//上下出=2
IF Autoflow=1
	AND AutoStatus
	AND NOT(DisablePB[11])
	AND LS_S11_UpDownBack
	AND NOT(SOL_S11_UpDown)
	AND (MachineRunStatus AND NOT(IndexData[11].FinishFlag[11]) AND IndexData[11].FinishFlag[10] AND IndexData[11].OKFlag[10] AND NOT(IndexData[11].NGFlag[10])
	OR Rtrig_test.Q) THEN
	Autoflow:=2;
	Error_LS_S11_UpDownOut1:=FALSE;
END_IF;
TON1(In:=Autoflow=2 AND LS_S11_UpDownOut, PT:=t#500ms);
//檢查開始=3
IF Autoflow=2 AND TON1.Q THEN
	Autoflow:=3;
END_IF;
IF Autoflow=3 AND HMIPV_S11_CurrentValue<=HMISV_S11_MaxValue AND HMIPV_S11_CurrentValue>=HMISV_S11_MinValue THEN		//OK
	IndexData[11].OKFlag[11]:=TRUE;
	IndexData[11].NGFlag[11]:=FALSE;
	IndexData[11].ErrorLog[11]:=0;
END_IF;
IF Autoflow=3 AND (HMIPV_S11_CurrentValue>HMISV_S11_MaxValue OR HMIPV_S11_CurrentValue<HMISV_S11_MinValue) THEN		//NG
	Error_LS_S11_UpDownOut1:=TRUE;
	IndexData[11].OKFlag[11]:=FALSE;
	IndexData[11].NGFlag[11]:=TRUE;
	IndexData[11].ErrorLog[11]:=3;
	BatchIndexCount:=BatchIndexCount-1;
END_IF;
TON2(In:=Autoflow=3 AND IndexData[11].FinishFlag[11], PT:=t#1000ms);
//上下回=4
IF Autoflow=3 AND TON2.Q AND (Rtrig_test.Q OR NOT(StepMode)) THEN
	Autoflow:=4;
END_IF;

//*************************************************************************
//手動
//上下電磁閥
R_TRIG_1[0](CLK:=HMIPB_SOL_S11_UpDown AND NOT(AutoStatus));
interlockback[0]:=TRUE;
interlockout[0]:=SNR_Index AND NOT(RY_Index);
(*SET*)
IF ((R_TRIG_1[0].Q AND NOT(solstatus[0])) OR Autoflow=2) AND interlockout[0] THEN
	SOL_S11_UpDown:=TRUE;
END_IF;
(*RESET*)
IF ((R_TRIG_1[0].Q AND (solstatus[0])) OR Autoflow=4 OR Initflow=4) AND interlockback[0] THEN
	SOL_S11_UpDown:=FALSE;
END_IF;
(*STATUS*)
solstatus[0]:=SOL_S11_UpDown;

//標準值設定
IF HMIPB_S11_StandarValueSet THEN
	HMISV_S11_StandarValue:=HMIPV_S11_CurrentValue;
END_IF;

HMISV_S11_MaxValue:=HMISV_S11_StandarValue+HMISV_S11_PValue;	//最大值
HMISV_S11_MinValue:=HMISV_S11_StandarValue-HMISV_S11_NValue;	//最小值

(*************************************************************************
程序名稱:第11站檢查上夾板RESET流程
作者:蔡相偉
版本,日期,版本資訊:
1.0.0		2017/11/22		初始版本

PowerOn=0
Idle=1
上下回=4
*************************************************************************)
//PowerOn=0
IF NOT(SystemReadyStatus) THEN
	Initflow:=0;
END_IF;

//Idle=1
IF Initflow=0 AND SystemReadyStatus THEN
	Initflow:=1;
END_IF;

IF Initflow=4 AND LS_S11_UpDownBack THEN
	Initflow:=1;
END_IF;

//上下回=4
F_TRIG_1(CLK:= ErrorStatus[11] OR Error_PB_Estop);
IF Initflow=1 AND (F_TRIG_1.Q OR Manual2AutoFlag) THEN
	Initflow:=4;
END_IF;

//*************************************************************************
//Cycle Time
//*************************************************************************
TON_CT(In:=AutoFlow>1, PT:=t#500s);
CycleTime[11]:=LINT_TO_DINT(TimeToSec( TON_CT.ET));
END_PROGRAM

PROGRAM prStation13
VAR
    interlockback : ARRAY[0..1] OF BOOL;
    interlockout : ARRAY[0..1] OF BOOL;
    solstatus : ARRAY[0..1] OF BOOL;
    R_TRIG_1 : ARRAY[0..1] OF R_TRIG;
    Rtrig_test : R_TRIG;
    F_TRIG_1 : F_TRIG;
    Autoflow : INT;
    Initflow : INT;
    TON1 : TON;
    TON2 : TON;
    tPressTime : TIME;
    TON_CT : TON;
END_VAR
VAR_EXTERNAL
    IndexData : ARRAY[0..19] OF stIndexData;
    DisablePB : ARRAY[0..19] OF BOOL;
    SystemReadyStatus : BOOL;
    AutoStatus : BOOL;
    ErrorStatus : ARRAY[0..19] OF BOOL;
    Error_PB_EStop : BOOL;
    LS_S13_UpDownBack : BOOL;
    MachineRunStatus : BOOL;
    LS_S13_UpDownOut : BOOL;
    HMIPB_SOL_S13_UpDown : BOOL;
    SNR_Index : BOOL;
    RY_Index : BOOL;
    SOL_S13_UpDown : BOOL;
    Manual2AutoFlag : BOOL;
    TestPB : ARRAY[0..19] OF BOOL;
    LS_S13_TempHighWarring : BOOL;
    LS_S13_TempLowWarring : BOOL;
    Error_LS_S13_TempHighWarring : BOOL;
    Error_LS_S13_TempLowWarring : BOOL;
    HMISV_S13_PressTime : DINT;
    CycleTime : ARRAY[0..19] OF DINT;
    BatchIndexCount : DINT;
    Error_LS_S11_UpDownOut1 : BOOL;
    Error_LS_S13_UpDownOut1 : BOOL;
    StepMode : BOOL;
END_VAR
(*************************************************************************
程序名稱:第13站壓合流程
作者:蔡相偉
版本,日期,版本資訊:
1.0.0		2017/11/22		初始版本

PowerOn=0
Idle=1
上下出=2
檢查開始=3
上下回=4
*************************************************************************)
(*************************************************************************
異常碼
急停=1
氣缸=2
檢查NG=3
*************************************************************************)
//*************************************************************************
//本站狀態判斷
IF IndexData[13].OKFlag[13]
	OR IndexData[13].NGFlag[13] THEN
	IndexData[13].FinishFlag[13]:=TRUE;
END_IF;
//前站狀態判斷
IF  	IndexData[13].NGFlag[11] THEN
	IndexData[13].NGFlag[11]:=TRUE;
END_IF;
//本站關閉判斷
IF DisablePB[13] AND IndexData[13].FinishFlag[11] AND IndexData[13].OKFlag[11] AND NOT(IndexData[13].NGFlag[11]) THEN
	IndexData[13].OKFlag[13]:=TRUE;
END_IF;

Rtrig_test(CLK:=TestPB[13]);
//PowerOn=0
IF NOT(SystemReadyStatus AND AutoStatus AND NOT(ErrorStatus[13]) AND NOT(Error_PB_EStop)) THEN
	Autoflow:=0;
END_IF;
	//EStop異常碼
	IF Error_PB_Estop AND NOT(IndexData[13].FinishFlag[13]) AND IndexData[13].OkFlag[1] THEN
		IndexData[13].NGFlag[13]:=TRUE;
		IndexData[13].ErrorLog[13]:=1;
		BatchIndexCount:=BatchIndexCount-1;
	END_IF;
	//Error異常碼
	IF ErrorStatus[13] AND NOT(IndexData[13].FinishFlag[13]) AND IndexData[13].OkFlag[1] THEN
		IndexData[13].NGFlag[13]:=TRUE;
		IndexData[13].ErrorLog[13]:=2;
		BatchIndexCount:=BatchIndexCount-1;
	END_IF;
//Idle=1
IF AutoFlow=0 AND SystemReadyStatus AND AutoStatus AND NOT(ErrorStatus[13]) AND NOT(Error_PB_EStop) THEN
	AutoFlow:=1;
END_IF;

IF Autoflow=4 AND LS_S13_UpDownBack THEN
	Autoflow:=1;
END_IF;

//上下出=2
IF Autoflow=1
	AND AutoStatus
	AND NOT(DisablePB[13])
	AND LS_S13_UpDownBack
	AND NOT(SOL_S13_UpDown)
	AND NOT(Error_LS_S13_TempHighWarring)
	AND NOT(Error_LS_S13_TempLowWarring)
	AND (MachineRunStatus AND NOT(IndexData[13].FinishFlag[13]) AND IndexData[13].FinishFlag[11] AND IndexData[13].OKFlag[11] AND NOT(IndexData[13].NGFlag[11])
	OR Rtrig_test.Q) THEN
	Autoflow:=2;
	Error_LS_S13_UpDownOut1:=FALSE;
END_IF;

//檢查開始=3
IF Autoflow=2 AND NOT(LS_S13_UpDownBack) THEN
	Autoflow:=3;
END_IF;
tPressTime:=NanoSecToTime(HMISV_S13_PressTime*100000000);	//Define
TON1(In:=Autoflow=3 AND LS_S13_UpDownOut, PT:=tPressTime);		//OK
TON2(In:=NOT(TON1.Q), PT:=t#2s);		//NG
//上下回=4
IF Autoflow=3 AND TON1.Q AND (Rtrig_test.Q OR NOT(StepMode)) THEN
	IndexData[13].OKFlag[13]:=TRUE;
	IndexData[13].NGFlag[13]:=FALSE;
	IndexData[13].ErrorLog[13]:=0;
	Autoflow:=4;
END_IF;

IF Autoflow=3 AND TON2.Q AND (Rtrig_test.Q OR NOT(StepMode)) THEN
	Error_LS_S13_UpDownOut1:=TRUE;
	IndexData[13].OKFlag[13]:=FALSE;
	IndexData[13].NGFlag[13]:=TRUE;
	IndexData[13].ErrorLog[13]:=3;
	BatchIndexCount:=BatchIndexCount-1;
	Autoflow:=4;
END_IF;

//*************************************************************************
//手動
//上下電磁閥
R_TRIG_1[0](CLK:=HMIPB_SOL_S13_UpDown AND NOT(AutoStatus));
interlockback[0]:=TRUE;
interlockout[0]:=SNR_Index AND NOT(RY_Index);
(*SET*)
IF ((R_TRIG_1[0].Q AND NOT(solstatus[0])) OR Autoflow=2) AND interlockout[0] THEN
	SOL_S13_UpDown:=TRUE;
END_IF;
(*RESET*)
IF ((R_TRIG_1[0].Q AND (solstatus[0])) OR Autoflow=4 OR Initflow=4) AND interlockback[0] THEN
	SOL_S13_UpDown:=FALSE;
END_IF;
(*STATUS*)
solstatus[0]:=SOL_S13_UpDown;
(*************************************************************************
程序名稱:第13站壓合RESET流程
作者:蔡相偉
版本,日期,版本資訊:
1.0.0		2017/11/22		初始版本

PowerOn=0
Idle=1
上下回=4
*************************************************************************)
//PowerOn=0
IF NOT(SystemReadyStatus) THEN
	Initflow:=0;
END_IF;

//Idle=1
IF Initflow=0 AND SystemReadyStatus THEN
	Initflow:=1;
END_IF;

IF Initflow=4 AND LS_S13_UpDownBack THEN
	Initflow:=1;
END_IF;

//上下回=4
F_TRIG_1(CLK:= ErrorStatus[13] OR Error_PB_Estop);
IF Initflow=1 AND (F_TRIG_1.Q OR Manual2AutoFlag) THEN
	Initflow:=4;
END_IF;

//*************************************************************************
//Cycle Time
//*************************************************************************
TON_CT(In:=AutoFlow>1, PT:=t#500s);
CycleTime[13]:=LINT_TO_DINT(TimeToSec( TON_CT.ET));
END_PROGRAM

PROGRAM prStation15
VAR
    interlockback : ARRAY[0..1] OF BOOL;
    interlockout : ARRAY[0..1] OF BOOL;
    solstatus : ARRAY[0..1] OF BOOL;
    R_TRIG_1 : ARRAY[0..1] OF R_TRIG;
    Rtrig_test : R_TRIG;
    F_TRIG_1 : F_TRIG;
    Autoflow : INT;
    Initflow : INT;
    TON1 : TON;
    TON2 : TON;
    TON_CT : TON;
END_VAR
VAR_EXTERNAL
    IndexData : ARRAY[0..19] OF stIndexData;
    DisablePB : ARRAY[0..19] OF BOOL;
    SystemReadyStatus : BOOL;
    AutoStatus : BOOL;
    ErrorStatus : ARRAY[0..19] OF BOOL;
    Error_PB_EStop : BOOL;
    MachineRunStatus : BOOL;
    SNR_Index : BOOL;
    RY_Index : BOOL;
    Manual2AutoFlag : BOOL;
    TestPB : ARRAY[0..19] OF BOOL;
    HMIPB_SOL_S15_UpDown : BOOL;
    SOL_S15_UpDown : BOOL;
    HMISV_S15_StandarValue : DINT;
    HMIPV_S15_CurrentValue : DINT;
    HMISV_S15_MaxValue : DINT;
    HMISV_S15_PValue : DINT;
    HMISV_S15_MinValue : DINT;
    HMISV_S15_NValue : DINT;
    HMIPB_S15_StandarValueSet : BOOL;
    LS_S15_UpDownBack : BOOL;
    LS_S15_UpDownOut : BOOL;
    CycleTime : ARRAY[0..19] OF DINT;
    BatchIndexCount : DINT;
    Error_LS_S13_UpDownOut1 : BOOL;
    Error_LS_S15_UpDownOut1 : BOOL;
    StepMode : BOOL;
END_VAR
(*************************************************************************
程序名稱:第15站檢查壓合流程
作者:蔡相偉
版本,日期,版本資訊:
1.0.0		2017/11/28		初始版本

PowerOn=0
Idle=1
上下出=2
檢查開始=3
上下回=4
*************************************************************************)
(*************************************************************************
異常碼
急停=1
氣缸=2
檢查NG=3
*************************************************************************)
//*************************************************************************
//本站狀態判斷
IF IndexData[15].OKFlag[15]
	OR IndexData[15].NGFlag[15] THEN
	IndexData[15].FinishFlag[15]:=TRUE;
END_IF;
//前站狀態判斷
IF  	IndexData[15].NGFlag[13] THEN
	IndexData[15].NGFlag[13]:=TRUE;
END_IF;
//本站關閉判斷
IF DisablePB[15] AND IndexData[15].FinishFlag[13] AND IndexData[15].OKFlag[13] AND NOT(IndexData[15].NGFlag[13]) THEN
	IndexData[15].OKFlag[15]:=TRUE;
END_IF;

Rtrig_test(CLK:=TestPB[15]);
//PowerOn=0
IF NOT(SystemReadyStatus AND AutoStatus AND NOT(ErrorStatus[15]) AND NOT(Error_PB_EStop)) THEN
	Autoflow:=0;
END_IF;
	//EStop異常碼
	IF Error_PB_Estop AND NOT(IndexData[15].FinishFlag[15]) AND IndexData[15].OkFlag[1] THEN
		IndexData[15].NGFlag[15]:=TRUE;
		IndexData[15].ErrorLog[15]:=1;
		BatchIndexCount:=BatchIndexCount-1;
	END_IF;
	//Error異常碼
	IF ErrorStatus[15] AND NOT(IndexData[15].FinishFlag[15]) AND IndexData[15].OkFlag[1] THEN
		IndexData[15].NGFlag[15]:=TRUE;
		IndexData[15].ErrorLog[15]:=2;
		BatchIndexCount:=BatchIndexCount-1;
	END_IF;
//Idle=1
IF AutoFlow=0 AND SystemReadyStatus AND AutoStatus AND NOT(ErrorStatus[15]) AND NOT(Error_PB_EStop) THEN
	AutoFlow:=1;
END_IF;

IF Autoflow=4 AND LS_S15_UpDownBack THEN
	Autoflow:=1;
END_IF;

//上下出=2
IF Autoflow=1
	AND AutoStatus
	AND NOT(DisablePB[15])
	AND LS_S15_UpDownBack
	AND NOT(SOL_S15_UpDown)
	AND (MachineRunStatus AND NOT(IndexData[15].FinishFlag[15]) AND IndexData[15].FinishFlag[13] AND IndexData[15].OKFlag[13] AND NOT(IndexData[15].NGFlag[13])
	OR Rtrig_test.Q) THEN
	Autoflow:=2;
	Error_LS_S15_UpDownOut1:=FALSE;
END_IF;
TON1(In:=Autoflow=2 AND LS_S15_UpDownOut, PT:=t#500ms);
//檢查開始=3
IF Autoflow=2 AND TON1.Q THEN
	Autoflow:=3;
END_IF;
IF Autoflow=3 AND NOT(IndexData[15].FinishFlag[15]) AND HMIPV_S15_CurrentValue<=HMISV_S15_MaxValue AND HMIPV_S15_CurrentValue>=HMISV_S15_MinValue THEN		//OK
	IndexData[15].OKFlag[15]:=TRUE;
	IndexData[15].NGFlag[15]:=FALSE;
	IndexData[15].ErrorLog[15]:=0;
END_IF;
IF Autoflow=3 AND NOT(IndexData[15].FinishFlag[15]) AND (HMIPV_S15_CurrentValue>HMISV_S15_MaxValue OR HMIPV_S15_CurrentValue<HMISV_S15_MinValue) THEN		//NG
	Error_LS_S15_UpDownOut1:=TRUE;
	IndexData[15].OKFlag[15]:=FALSE;
	IndexData[15].NGFlag[15]:=TRUE;
	IndexData[15].ErrorLog[15]:=3;
	BatchIndexCount:=BatchIndexCount-1;
END_IF;
TON2(In:=Autoflow=3 AND IndexData[15].FinishFlag[15], PT:=t#1000ms);
//上下回=4
IF Autoflow=3 AND TON2.Q AND (Rtrig_test.Q OR NOT(StepMode)) THEN
	Autoflow:=4;
END_IF;

//*************************************************************************
//手動
//上下電磁閥
R_TRIG_1[0](CLK:=HMIPB_SOL_S15_UpDown AND NOT(AutoStatus));
interlockback[0]:=TRUE;
interlockout[0]:=SNR_Index AND NOT(RY_Index);
(*SET*)
IF ((R_TRIG_1[0].Q AND NOT(solstatus[0])) OR Autoflow=2) AND interlockout[0] THEN
	SOL_S15_UpDown:=TRUE;
END_IF;
(*RESET*)
IF ((R_TRIG_1[0].Q AND (solstatus[0])) OR Autoflow=4 OR Initflow=4) AND interlockback[0] THEN
	SOL_S15_UpDown:=FALSE;
END_IF;
(*STATUS*)
solstatus[0]:=SOL_S15_UpDown;

//標準值設定
IF HMIPB_S15_StandarValueSet THEN
	HMISV_S15_StandarValue:=HMIPV_S15_CurrentValue;
END_IF;

HMISV_S15_MaxValue:=HMISV_S15_StandarValue+HMISV_S15_PValue;	//最大值
HMISV_S15_MinValue:=HMISV_S15_StandarValue-HMISV_S15_NValue;	//最小值

(*************************************************************************
程序名稱:第15站檢查壓合RESET流程
作者:蔡相偉
版本,日期,版本資訊:
1.0.0		2017/11/22		初始版本

PowerOn=0
Idle=1
上下回=4
*************************************************************************)
//PowerOn=0
IF NOT(SystemReadyStatus) THEN
	Initflow:=0;
END_IF;

//Idle=1
IF Initflow=0 AND SystemReadyStatus THEN
	Initflow:=1;
END_IF;

IF Initflow=4 AND LS_S15_UpDownBack THEN
	Initflow:=1;
END_IF;

//上下回=4
F_TRIG_1(CLK:= ErrorStatus[15] OR Error_PB_Estop);
IF Initflow=1 AND (F_TRIG_1.Q OR Manual2AutoFlag) THEN
	Initflow:=4;
END_IF;

//*************************************************************************
//Cycle Time
//*************************************************************************
TON_CT(In:=AutoFlow>1, PT:=t#500s);
CycleTime[15]:=LINT_TO_DINT(TimeToSec( TON_CT.ET));
END_PROGRAM

PROGRAM prStation16
VAR
    AutoFlow : INT;
    Rtrig_test : R_TRIG;
    Rtrig_test2 : R_TRIG;
    TON_CT : TON;
END_VAR
VAR_EXTERNAL
    IndexData : ARRAY[0..19] OF stIndexData;
    DisablePB : ARRAY[0..19] OF BOOL;
    TestPB : ARRAY[0..19] OF BOOL;
    SystemReadyStatus : BOOL;
    ErrorStatus : ARRAY[0..19] OF BOOL;
    Error_PB_EStop : BOOL;
    AutoStatus : BOOL;
    MachineRunStatus : BOOL;
    HMIPB_YAMAHA_Unload_OKStart : BOOL;
    YAMAHA_Unload_OKStart : BOOL;
    YAMAHA_Unload_Finish : BOOL;
    HMIPB_YAMAHA_Unload_NGStart : BOOL;
    YAMAHA_Unload_NGStart : BOOL;
    CycleTime : ARRAY[0..19] OF DINT;
    BatchOKCount : DINT;
    BatchIndexCount : DINT;
    BatchNGCount : DINT;
END_VAR
(*
程序名稱:第16站下料流程
作者:蔡相偉
版本,日期,版本資訊:
1.0.0		2017/11/21		初始版本
PowerOn=0
Idle=1|--->OK下料開始=10--->OK下料完成=11
		  |--->NG下料開始=20--->NG下料完成=21
*)
//本站狀態判斷
IF IndexData[16].OKFlag[16]
	OR IndexData[16].NGFlag[16] THEN
	IndexData[16].FinishFlag[16]:=TRUE;
END_IF;

//前站狀態判斷
IF NOT(IndexData[16].OKFlag[1]) THEN
	IndexData[16].NGFlag[16]:=TRUE;
END_IF;

(*
//本站關閉判斷
IF DisablePB[1] THEN
	IndexData[1].NGFlag[1]:=TRUE;
END_IF;
*)
Rtrig_test(CLK:=HMIPB_YAMAHA_Unload_OKStart);
Rtrig_test2(CLK:=HMIPB_YAMAHA_Unload_NGStart);
//PowerOn=0
IF NOT(SystemReadyStatus AND AutoStatus AND NOT(ErrorStatus[16]) AND NOT(Error_PB_EStop)) THEN
	Autoflow:=0;
END_IF;

//Idle=1
IF AutoFlow=0 AND SystemReadyStatus AND AutoStatus AND NOT(ErrorStatus[16]) AND NOT(Error_PB_EStop) THEN
	AutoFlow:=1;
END_IF;

IF AutoFlow=11 AND NOT(YAMAHA_Unload_OKStart) AND IndexData[16].FinishFlag[16] THEN
	AutoFlow:=1;
END_IF;

IF AutoFlow=21 AND NOT(YAMAHA_Unload_NGStart) AND IndexData[16].FinishFlag[16] THEN
	AutoFlow:=1;
END_IF;

//OK下料開始=10
IF Autoflow=1
	AND AutoStatus
	AND NOT(DisablePB[16])
	AND (MachineRunStatus AND NOT(IndexData[16].FinishFlag[16]) AND IndexData[16].OKFlag[1] AND IndexData[16].FinishFlag[15] AND IndexData[16].OKFlag[15] AND NOT(IndexData[16].NGFlag[15]) OR Rtrig_test.Q) THEN
	Autoflow:=10;
END_IF;
IF AutoFlow=10 THEN
	YAMAHA_Unload_OKStart:=TRUE;
END_IF;
IF YAMAHA_Unload_Finish OR AutoFlow=0 THEN
	YAMAHA_Unload_OKStart:=FALSE;
END_IF;

//OK下料完成=11
IF AutoFlow=10 AND (YAMAHA_Unload_Finish) THEN
	BatchOKCount:=BatchOKCount+1;
	BatchIndexCount:=BatchIndexCount-1;
	AutoFlow:=11;
END_IF;
IF AutoFlow=11 THEN
	IndexData[16].OKFlag[16]:=TRUE;
END_IF;

//NG下料開始=20
IF Autoflow=1
	AND AutoStatus
	AND NOT(DisablePB[16])
	AND (MachineRunStatus AND NOT(IndexData[16].FinishFlag[16]) AND IndexData[16].OKFlag[1] AND IndexData[16].FinishFlag[15] AND (IndexData[16].NGFlag[15]) OR Rtrig_test2.Q) THEN
	Autoflow:=20;
END_IF;
IF AutoFlow=20 THEN
	YAMAHA_Unload_NGStart:=TRUE;
END_IF;
IF YAMAHA_Unload_Finish OR AutoFlow=0 THEN
	YAMAHA_Unload_NGStart:=FALSE;
END_IF;

//NG下料完成=21
IF AutoFlow=20 AND (YAMAHA_Unload_Finish) THEN
	BatchNGCount:=BatchNGCount+1;
	BatchIndexCount:=BatchIndexCount-1;
	AutoFlow:=21;
END_IF;
IF AutoFlow=21 THEN
	IndexData[16].NGFlag[16]:=TRUE;
END_IF;

//*************************************************************************
//Cycle Time
//*************************************************************************
TON_CT(In:=AutoFlow>1, PT:=t#500s);
CycleTime[16]:=LINT_TO_DINT(TimeToSec( TON_CT.ET));
END_PROGRAM

PROGRAM prFeedAndSupplier
VAR
    Supplier_S6 : fbFull;
    Supplier_S8 : fbFull;
    Supplier_S10 : fbFull;
    Feeder_S6 : fbFeed;
    Feeder_S8 : fbFeed;
    Feeder_S10 : fbFeed;
END_VAR
VAR_EXTERNAL
    SNR_S6_Full : BOOL;
    RY_S6_Full : BOOL;
    Error_SNR_S6_Full : BOOL;
    FullNotExistTime : ARRAY[0..19] OF DINT;
    FullExistTime : ARRAY[0..19] OF DINT;
    FullNotExistErrorTime : ARRAY[0..19] OF DINT;
    SNR_S8_Full : BOOL;
    RY_S8_Full : BOOL;
    Error_SNR_S8_Full : BOOL;
    SNR_S10_Full : BOOL;
    RY_S10_Full : BOOL;
    Error_SNR_S10_Full : BOOL;
    FeedStart : ARRAY[0..19] OF BOOL;
    PB_Reset : BOOL;
    FeedFinish : ARRAY[0..19] OF BOOL;
    Error_LS_S6_THBack : BOOL;
    Error_LS_S6_THOut : BOOL;
    LS_S6_UpDownBack : BOOL;
    SOL_S6_UpDown : BOOL;
    LS_S6_MoveBack : BOOL;
    SNR_S6_Feed : BOOL;
    LS_S6_THBack : BOOL;
    LS_S6_THOut : BOOL;
    HMIPB_SOL_S6_TH : BOOL;
    FeedNotExistTime : ARRAY[0..19] OF DINT;
    FeedExistTime : ARRAY[0..19] OF DINT;
    Error_SNR_S6_Feed : BOOL;
    RY_S6_Feed : BOOL;
    SOL_S6_TH : BOOL;
    Error_LS_S8_THBack : BOOL;
    Error_LS_S8_THOut : BOOL;
    LS_S8_UpDownBack : BOOL;
    SOL_S8_UpDown : BOOL;
    LS_S8_MoveBack : BOOL;
    SNR_S8_Feed : BOOL;
    LS_S8_THBack : BOOL;
    LS_S8_THOut : BOOL;
    HMIPB_SOL_S8_TH : BOOL;
    Error_SNR_S8_Feed : BOOL;
    RY_S8_Feed : BOOL;
    SOL_S8_TH : BOOL;
    Error_LS_S10_THBack : BOOL;
    Error_LS_S10_THOut : BOOL;
    LS_S10_UpDownBack : BOOL;
    SOL_S10_UpDown : BOOL;
    LS_S10_MoveBack : BOOL;
    SNR_S10_Feed : BOOL;
    LS_S10_THBack : BOOL;
    LS_S10_THOut : BOOL;
    HMIPB_SOL_S10_TH : BOOL;
    Error_SNR_S10_Feed : BOOL;
    RY_S10_Feed : BOOL;
    SOL_S10_TH : BOOL;
    Manual2AutoFlag : BOOL;
END_VAR
//第6站振動筒
Supplier_S6();
Supplier_S6.bFullSNR:=SNR_S6_Full;
Supplier_S6.iItemNotExistDelayTime:=FullNotExistTime[6];
Supplier_S6.iItemExistTime:=FullExistTime[6];
Supplier_S6.iItemNotExistErrorTime:=FullNotExistErrorTime[6];
RY_S6_Full:=Supplier_S6.bFullRY;
Error_SNR_S6_Full:=Supplier_S6.bFullSNRError;

//第8站振動筒
Supplier_S8();
Supplier_S8.bFullSNR:=SNR_S8_Full;
Supplier_S8.iItemNotExistDelayTime:=FullNotExistTime[8];
Supplier_S8.iItemExistTime:=FullExistTime[8];
Supplier_S8.iItemNotExistErrorTime:=FullNotExistErrorTime[8];
RY_S8_Full:=Supplier_S8.bFullRY;
Error_SNR_S8_Full:=Supplier_S8.bFullSNRError;

//第10站振動筒
Supplier_S10();
Supplier_S10.bFullSNR:=SNR_S10_Full;
Supplier_S10.iItemNotExistDelayTime:=FullNotExistTime[10];
Supplier_S10.iItemExistTime:=FullExistTime[10];
Supplier_S10.iItemNotExistErrorTime:=FullNotExistErrorTime[10];
RY_S10_Full:=Supplier_S10.bFullRY;
Error_SNR_S10_Full:=Supplier_S10.bFullSNRError;

//第6站平送
Feeder_S6();
Feeder_S6.bErrorTHBack:=Error_LS_S6_THBack;
Feeder_S6.bErrorTHOut:=Error_LS_S6_THOut;
Feeder_S6.bFeedStart:=FeedStart[6] OR Manual2AutoFlag;
Feeder_S6.bInterlock_thback:=(LS_S6_UpDownBack AND NOT(SOL_S6_UpDown)) OR NOT(LS_S6_MoveBack);
Feeder_S6.bInterlock_thout:=(LS_S6_UpDownBack AND NOT(SOL_S6_UpDown)) OR NOT(LS_S6_MoveBack);
Feeder_S6.bObjSNR:=SNR_S6_Feed;
Feeder_S6.bReset:=PB_Reset;
Feeder_S6.bSupplierRY:=RY_S6_Full;
Feeder_S6.bTHBackLS:=LS_S6_THBack;
Feeder_S6.bTHOutLS:=LS_S6_THOut;
Feeder_S6.bTHPB:=HMIPB_SOL_S6_TH;
Feeder_S6.wNoObjDelayTime:=FeedNotExistTime[6];
Feeder_S6.wObjectExistDelayTime:=FeedExistTime[6];
Error_SNR_S6_Feed :=Feeder_S6.bFeedError;
FeedFinish[6]:= Feeder_S6.bFeedFinish;
RY_S6_Feed:= Feeder_S6.bFeedRY;
SOL_S6_TH:= Feeder_S6.bTHSOL;

//第8站平送
Feeder_S8();
Feeder_S8.bErrorTHBack:=Error_LS_S8_THBack;
Feeder_S8.bErrorTHOut:=Error_LS_S8_THOut;
Feeder_S8.bFeedStart:=FeedStart[8] OR Manual2AutoFlag;
Feeder_S8.bInterlock_thback:=(LS_S8_UpDownBack AND NOT(SOL_S8_UpDown)) OR NOT(LS_S8_MoveBack);
Feeder_S8.bInterlock_thout:=(LS_S8_UpDownBack AND NOT(SOL_S8_UpDown)) OR NOT(LS_S8_MoveBack);
Feeder_S8.bObjSNR:=SNR_S8_Feed;
Feeder_S8.bReset:=PB_Reset;
Feeder_S8.bSupplierRY:=RY_S8_Full;
Feeder_S8.bTHBackLS:=LS_S8_THBack;
Feeder_S8.bTHOutLS:=LS_S8_THOut;
Feeder_S8.bTHPB:=HMIPB_SOL_S8_TH;
Feeder_S8.wNoObjDelayTime:=FeedNotExistTime[8];
Feeder_S8.wObjectExistDelayTime:=FeedExistTime[8];
Error_SNR_S8_Feed:=Feeder_S8.bFeedError;
FeedFinish[8]:= Feeder_S8.bFeedFinish;
RY_S8_Feed:= Feeder_S8.bFeedRY;
SOL_S8_TH:= Feeder_S8.bTHSOL;

//第10站平送
Feeder_S10();
Feeder_S10.bErrorTHBack:=Error_LS_S10_THBack;
Feeder_S10.bErrorTHOut:=Error_LS_S10_THOut;
Feeder_S10.bFeedStart:=FeedStart[10] OR Manual2AutoFlag;
Feeder_S10.bInterlock_thback:=(LS_S10_UpDownBack AND NOT(SOL_S10_UpDown)) OR NOT(LS_S10_MoveBack);
Feeder_S10.bInterlock_thout:=(LS_S10_UpDownBack AND NOT(SOL_S10_UpDown)) OR NOT(LS_S10_MoveBack);
Feeder_S10.bObjSNR:=SNR_S10_Feed;
Feeder_S10.bReset:=PB_Reset;
Feeder_S10.bSupplierRY:=RY_S10_Full;
Feeder_S10.bTHBackLS:=LS_S10_THBack;
Feeder_S10.bTHOutLS:=LS_S10_THOut;
Feeder_S10.bTHPB:=HMIPB_SOL_S10_TH;
Feeder_S10.wNoObjDelayTime:=FeedNotExistTime[10];
Feeder_S10.wObjectExistDelayTime:=FeedExistTime[10];
Error_SNR_S10_Feed:=Feeder_S10.bFeedError;
FeedFinish[10]:= Feeder_S10.bFeedFinish;
RY_S10_Feed:= Feeder_S10.bFeedRY;
SOL_S10_TH:= Feeder_S10.bTHSOL;
END_PROGRAM

PROGRAM prNGCount
VAR
    R_TRIG1 : ARRAY[0..19] OF R_TRIG;
    iCount : ARRAY[0..19] OF INT;
END_VAR
VAR_EXTERNAL
    IndexData : ARRAY[0..19] OF stIndexData;
    Error_NGCount : ARRAY[0..19] OF BOOL;
    PB_Reset : BOOL;
    HMIPB_PB_Reset : BOOL;
END_VAR
//Over 3 times NG S2
R_TRIG1[0](Clk:=IndexData[2].NGFlag[2]);
IF IndexData[2].OKFlag[1] AND R_TRIG1[0].Q THEN
	iCount[2]:=iCount[2]+1;
END_IF;
IF IndexData[2].OKFlag[2] THEN
	iCount[2]:=0;
END_IF;
IF iCount[2]>=3 THEN
	Error_NGCount[2]:=TRUE;
ELSE
	Error_NGCount[2]:=FALSE;
END_IF;
IF PB_Reset OR HMIPB_PB_Reset THEN
	iCount[2]:=0;
END_IF;

//Over 3 times NG S4
R_TRIG1[1](Clk:=IndexData[4].NGFlag[4]);
IF IndexData[4].OKFlag[1] AND R_TRIG1[1].Q THEN
	iCount[4]:=iCount[4]+1;
END_IF;
IF IndexData[4].OKFlag[4] THEN
	iCount[4]:=0;
END_IF;
IF iCount[4]>=3 THEN
	Error_NGCount[4]:=TRUE;
ELSE
	Error_NGCount[4]:=FALSE;
END_IF;
IF PB_Reset OR HMIPB_PB_Reset THEN
	iCount[4]:=0;
END_IF;

//Over 3 times NG S5
R_TRIG1[2](Clk:=IndexData[5].NGFlag[5]);
IF IndexData[5].OKFlag[1] AND R_TRIG1[2].Q THEN
	iCount[5]:=iCount[5]+1;
END_IF;
IF IndexData[5].OKFlag[5] THEN
	iCount[5]:=0;
END_IF;
IF iCount[5]>=3 THEN
	Error_NGCount[5]:=TRUE;
ELSE
	Error_NGCount[5]:=FALSE;
END_IF;
IF PB_Reset OR HMIPB_PB_Reset THEN
	iCount[5]:=0;
END_IF;

//Over 3 times NG S6
R_TRIG1[3](Clk:=IndexData[6].NGFlag[6]);
IF IndexData[6].OKFlag[1] AND R_TRIG1[3].Q THEN
	iCount[6]:=iCount[6]+1;
END_IF;
IF IndexData[6].OKFlag[6] THEN
	iCount[6]:=0;
END_IF;
IF iCount[6]>=3 THEN
	Error_NGCount[6]:=TRUE;
ELSE
	Error_NGCount[6]:=FALSE;
END_IF;
IF PB_Reset OR HMIPB_PB_Reset THEN
	iCount[6]:=0;
END_IF;

//Over 3 times NG S7
R_TRIG1[4](Clk:=IndexData[7].NGFlag[7]);
IF IndexData[7].OKFlag[1] AND R_TRIG1[4].Q THEN
	iCount[7]:=iCount[7]+1;
END_IF;
IF IndexData[7].OKFlag[7] THEN
	iCount[7]:=0;
END_IF;
IF iCount[7]>=3 THEN
	Error_NGCount[7]:=TRUE;
ELSE
	Error_NGCount[7]:=FALSE;
END_IF;
IF PB_Reset OR HMIPB_PB_Reset THEN
	iCount[7]:=0;
END_IF;

//Over 3 times NG S8
R_TRIG1[5](Clk:=IndexData[8].NGFlag[8]);
IF IndexData[8].OKFlag[1] AND R_TRIG1[5].Q THEN
	iCount[8]:=iCount[8]+1;
END_IF;
IF IndexData[8].OKFlag[8] THEN
	iCount[8]:=0;
END_IF;
IF iCount[8]>=3 THEN
	Error_NGCount[8]:=TRUE;
ELSE
	Error_NGCount[8]:=FALSE;
END_IF;
IF PB_Reset OR HMIPB_PB_Reset THEN
	iCount[8]:=0;
END_IF;

//Over 3 times NG S9
R_TRIG1[6](Clk:=IndexData[9].NGFlag[9]);
IF IndexData[9].OKFlag[1] AND R_TRIG1[6].Q THEN
	iCount[9]:=iCount[9]+1;
END_IF;
IF IndexData[9].OKFlag[9] THEN
	iCount[9]:=0;
END_IF;
IF iCount[9]>=3 THEN
	Error_NGCount[9]:=TRUE;
ELSE
	Error_NGCount[9]:=FALSE;
END_IF;
IF PB_Reset OR HMIPB_PB_Reset THEN
	iCount[9]:=0;
END_IF;

//Over 3 times NG S10
R_TRIG1[7](Clk:=IndexData[10].NGFlag[10]);
IF IndexData[10].OKFlag[1] AND R_TRIG1[7].Q THEN
	iCount[10]:=iCount[10]+1;
END_IF;
IF IndexData[10].OKFlag[10] THEN
	iCount[10]:=0;
END_IF;
IF iCount[10]>=3 THEN
	Error_NGCount[10]:=TRUE;
ELSE
	Error_NGCount[10]:=FALSE;
END_IF;
IF PB_Reset OR HMIPB_PB_Reset THEN
	iCount[10]:=0;
END_IF;

//Over 3 times NG S11
R_TRIG1[8](Clk:=IndexData[11].NGFlag[11]);
IF IndexData[11].OKFlag[1] AND R_TRIG1[8].Q THEN
	iCount[11]:=iCount[11]+1;
END_IF;
IF IndexData[11].OKFlag[11] THEN
	iCount[11]:=0;
END_IF;
IF iCount[11]>=3 THEN
	Error_NGCount[11]:=TRUE;
ELSE
	Error_NGCount[11]:=FALSE;
END_IF;
IF PB_Reset OR HMIPB_PB_Reset THEN
	iCount[11]:=0;
END_IF;

//Over 3 times NG S13
R_TRIG1[9](Clk:=IndexData[13].NGFlag[13]);
IF IndexData[13].OKFlag[1] AND R_TRIG1[9].Q THEN
	iCount[13]:=iCount[13]+1;
END_IF;
IF IndexData[13].OKFlag[13] THEN
	iCount[13]:=0;
END_IF;
IF iCount[13]>=3 THEN
	Error_NGCount[13]:=TRUE;
ELSE
	Error_NGCount[13]:=FALSE;
END_IF;
IF PB_Reset OR HMIPB_PB_Reset THEN
	iCount[13]:=0;
END_IF;

//Over 3 times NG S15
R_TRIG1[10](Clk:=IndexData[15].NGFlag[15]);
IF IndexData[15].OKFlag[1] AND R_TRIG1[10].Q THEN
	iCount[15]:=iCount[15]+1;
END_IF;
IF IndexData[15].OKFlag[15] THEN
	iCount[15]:=0;
END_IF;
IF iCount[15]>=3 THEN
	Error_NGCount[15]:=TRUE;
ELSE
	Error_NGCount[15]:=FALSE;
END_IF;
IF PB_Reset OR HMIPB_PB_Reset THEN
	iCount[15]:=0;
END_IF;
END_PROGRAM

FUNCTION_BLOCK fbErrorDouble
VAR
    TON_1 : TON;
    TON_2 : TON;
END_VAR
VAR_INPUT
    bAutoStatus : BOOL;
    bResetPB : BOOL;
    bBackLS : BOOL;
    bOutLS : BOOL;
    bBackSOL : BOOL;
    bOutSOL : BOOL;
END_VAR
VAR_OUTPUT
    bErrorStatus_Back : BOOL;
    bErrorStatus_Out : BOOL;
END_VAR
IF bAutoStatus AND NOT(bResetPB) THEN
	(*歸磁簧開關*)
	TON_1(IN:=bBackSOL AND NOT(bBackLS), PT:=t#5s);
	IF TON_1.Q THEN
		bErrorStatus_Back:=TRUE;
	END_IF;
	(*出磁簧開關*)
	TON_2(IN:=bOutSOL AND NOT(bOutLS), PT:=t#5s);
	IF TON_2.Q THEN
		bErrorStatus_Out:=TRUE;
	END_IF;
END_IF;
IF bResetPB THEN
	bErrorStatus_Back:=FALSE;
	bErrorStatus_Out:=FALSE;
END_IF;
END_FUNCTION_BLOCK

FUNCTION_BLOCK fbErrorSingle
VAR
    TON_1 : TON;
    TON_2 : TON;
END_VAR
VAR_INPUT
    bAutoStatus : BOOL;
    bResetPB : BOOL;
    bSOL : BOOL;
    bBackLS : BOOL;
    bOutLS : BOOL;
END_VAR
VAR_OUTPUT
    bErrorStatus_Back : BOOL;
    bErrorStatus_Out : BOOL;
END_VAR
IF bAutoStatus AND NOT(bResetPB) THEN
	(*歸磁簧開關*)
	TON_1(IN:=(NOT(bSOL) AND NOT(bBackLS)) OR ((bSOL) AND bBackLS), PT:=t#5s);
	IF TON_1.Q THEN
		bErrorStatus_Back:=TRUE;
	END_IF;
	(*出磁簧開關*)
	TON_2(IN:=(NOT(bSOL) AND (bOutLS)) OR ((bSOL) AND NOT(bOutLS)), PT:=t#5s);
	IF TON_2.Q THEN
		bErrorStatus_Out:=TRUE;
	END_IF;
END_IF;
IF bResetPB THEN
	bErrorStatus_Back:=FALSE;
	bErrorStatus_Out:=FALSE;
END_IF;
END_FUNCTION_BLOCK

FUNCTION_BLOCK fbFull
VAR
    AutoFlow : INT;
    TON_Auto1 : TON;
    TON_Auto2 : TON;
    TON_Auto3 : TON;
    tItemNotExistDelayTime : TIME;
    tItemExistTime : TIME;
    tItemNotExistErrorTime : TIME;
END_VAR
VAR_INPUT
    bFullSNR : BOOL;
    iItemNotExistDelayTime : LINT;
    iItemExistTime : LINT;
    iItemNotExistErrorTime : LINT;
END_VAR
VAR_OUTPUT
    bFullRY : BOOL;
    bFullSNRError : BOOL;
END_VAR
VAR_EXTERNAL
    SystemReadyStatus : BOOL;
END_VAR
(******************************************************************
程式:振動筒程序
作者:蔡相偉
版本資訊:v1.0		2016/4/16
******************************************************************)
//時間轉換
tItemNotExistDelayTime:=NanoSecToTime(In:=iItemNotExistDelayTime*100000000);
tItemExistTime:=NanoSecToTime(In:=iItemExistTime*100000000);
tItemNotExistErrorTime:=NanoSecToTime(In:=iItemNotExistErrorTime*100000000);
(*流程*)
(*PowerOn=0*)
IF NOT(SystemReadyStatus) THEN
	AutoFlow:=0;
END_IF;

(*Idle=1*)
IF AutoFlow=0 AND SystemReadyStatus THEN
	AutoFlow:=1;
END_IF;

IF AutoFlow=3 THEN
	AutoFlow:=1;
END_IF;

(*振動筒起振=2*)
TON_Auto1(IN:=AutoFlow=1 AND NOT(bFullSNR) , PT:=tItemNotExistDelayTime);
IF AutoFlow=1 AND TON_Auto1.Q THEN
	AutoFlow:=2;
END_IF;

(*振動筒停振=3*)
TON_Auto2(IN:=AutoFlow=2 AND bFullSNR , PT:=tItemExistTime);
TON_Auto3(IN:=NOT(bFullSNR) AND bFullRY, PT:=tItemNotExistErrorTime);
IF AutoFlow=2 AND TON_Auto2.Q THEN
	AutoFlow:=3;
END_IF;
(******************************************************************)
(*輸出*)
(*振動筒繼電器*)
IF AutoFlow=2 THEN
	bFullRY:=TRUE;
	ELSE
	bFullRY:=FALSE;
END_IF;
(*振動筒滿料異常*)
IF AutoFlow=2 AND (TON_Auto3.Q) THEN
	bFullSNRError:=TRUE;
	ELSE
	bFullSNRError:=FALSE;
END_IF;
END_FUNCTION_BLOCK

FUNCTION_BLOCK fbFeed
VAR
    tNoObjDelayTime : TIME;
    tObjectExistDelayTime : TIME;
    Autoflow : INT;
    TON_1 : TON;
    TON_2 : TON;
    TON_3 : TON;
    ObjSNRStatus : BOOL;
    THStatus : BOOL;
    R_TRIG_1 : R_TRIG;
    R_TRIG_2 : R_TRIG;
    R_TRIG_3 : R_TRIG;
    R_TRIG_4 : R_TRIG;
END_VAR
VAR_INPUT
    wNoObjDelayTime : LINT;
    wObjectExistDelayTime : LINT;
    bReset : BOOL;
    bTHPB : BOOL;
    bObjSNR : BOOL;
    bFeedStart : BOOL;
    bTHBackLS : BOOL;
    bTHOutLS : BOOL;
    bErrorTHBack : BOOL;
    bErrorTHOut : BOOL;
    bInterlock_thback : BOOL;
    bInterlock_thout : BOOL;
    bSupplierRY : BOOL;
END_VAR
VAR_OUTPUT
    bFeedError : BOOL;
    bFeedFinish : BOOL;
    bTHSOL : BOOL;
    bFeedRY : BOOL;
END_VAR
VAR_EXTERNAL
    SystemReadyStatus : BOOL;
    AutoStatus : BOOL;
END_VAR
(*************************************************************************
程序名稱:平送FB
作者:蔡相偉
版本,日期,版本資訊:
1.0.0	2016/6/28		初始版本

PowerOn=0
Idle=1
無料,節流出=2
到出,平送起振=3
工件到位,平送停振=4
節流回=5
節流到回=6
*************************************************************************)
//時間轉換
tNoObjDelayTime:=NanoSecToTime(wNoObjDelayTime*100000000);
tObjectExistDelayTime:=NanoSecToTime(wObjectExistDelayTime*100000000);

//PowerOn=0
IF Autoflow=0 AND SystemReadyStatus AND NOT(bErrorTHBack) AND NOT(bErrorTHOut) AND AutoStatus  THEN
	Autoflow:=1;
END_IF;

(*Idle=1*)
TON_1(IN:= Autoflow=1 AND NOT(bObjSNR) ,PT:= tNoObjDelayTime);
IF Autoflow=1 AND (bFeedStart) THEN
	Autoflow:=2;
END_IF;
(*無料,節流出=2*)
IF Autoflow=2 THEN
	ObjSNRStatus:=FALSE;
END_IF;

IF Autoflow=2 AND bTHOutLS THEN
	Autoflow:=3;
END_IF;
(*到出,平送起振=3*)
IF Autoflow=3 AND bObjSNR THEN
	ObjSNRStatus:=TRUE;
END_IF;
TON_2(IN:= Autoflow=3 AND ObjSNRStatus ,PT:= tObjectExistDelayTime);
TON_3(IN:= Autoflow=3 AND NOT(ObjSNRStatus) ,PT:= t#4s);
IF TON_3.Q THEN
	bFeedError:=TRUE;
END_IF;
IF bReset THEN
	bFeedError:=FALSE;
END_IF;

IF Autoflow=3 AND TON_2.Q AND NOT(bFeedError) THEN
	Autoflow:=4;
END_IF;
(*工件到位,平送停振=4*)
IF Autoflow=4 THEN
	Autoflow:=5;
END_IF;
(*節流回=5*)
IF Autoflow=5 AND bTHBackLS THEN
	Autoflow:=6;
END_IF;
(*節流到回=6*)
IF Autoflow=6 THEN
	bFeedFinish:=TRUE;
	ELSE
	bFeedFinish:=FALSE;
END_IF;

IF Autoflow=6 AND NOT(bFeedStart) THEN
	Autoflow:=1;
END_IF;
(*************************************************************************)
(*Error*)
R_TRIG_3(CLK:=bErrorTHBack);
R_TRIG_4(CLK:=bErrorTHOut);

IF NOT(SystemReadyStatus) OR NOT(AutoStatus) OR bErrorTHBack OR bErrorTHOut THEN
	Autoflow:=0;
END_IF;

(*************************************************************************)
(*手動*)
(*節流*)
R_TRIG_1(CLK:=bTHPB AND NOT(AutoStatus));
(*SET*)
IF (((R_TRIG_1.Q) AND NOT(THStatus)) OR Autoflow=2 OR R_TRIG_3.Q) AND bInterlock_thout THEN
	bTHSOL:=TRUE;
END_IF;
(*RESET*)
IF (((R_TRIG_1.Q) AND THStatus) OR Autoflow=5 OR R_TRIG_4.Q) AND bInterlock_thback THEN
	bTHSOL:=FALSE;
END_IF;
(*STATE*)
THStatus:=bTHSOL;

(*平送*)
(*輸出*)
bFeedRY:=Autoflow=2 OR Autoflow=3 OR bSupplierRY OR bTHSOL;
END_FUNCTION_BLOCK